# EPICS substitutions: IOCs/MS_DAQ/iocBoot/iocMS/MS.substitutions
file "$(TOP)/db/MS.template"
{
pattern
{P,N,}
{MS:, 1,}
{MS:, 2,}
{MS:, 3,}
{MS:, 4,}
{MS:, 5,}
{MS:, 6,}
{MS:, 7,}
{MS:, 8,}
{MS:, 9,}
{MS:, 10,}
{MS:, 11,}
{MS:, 12,}
{MS:, 13,}
{MS:, 14,}
{MS:, 15,}
{MS:, 16,}
{MS:, 17,}
{MS:, 18,}
{MS:, 19,}
{MS:, 20,}
}
